TEXTLIST MachineType
  0 = 'None'
  1 = 'RH353'
  2 = 'RH367'
  3 = 'RH311'
  4 = 'RH201'
  5 = 'RH069'
  6 = 'RH373'
  7 = 'LH353'
  8 = 'LH367'
  9 = 'LH311'
  10 = 'LH201'
  11 = 'LH069'
  12 = 'LH373'
   = ''
END_TEXTLIST

(* stored: Version 1.1.0.1, ProductVersion 3.1.4024.3
   TextList MachineType: Id {52a7b924-6128-4d80-ace3-4eabc4fb45fe} *)
